// LS Electric XG5000 project: plc-assemble
// PLC LSPLC

PROGRAM NewProgram (task: 스캔 프로그램)

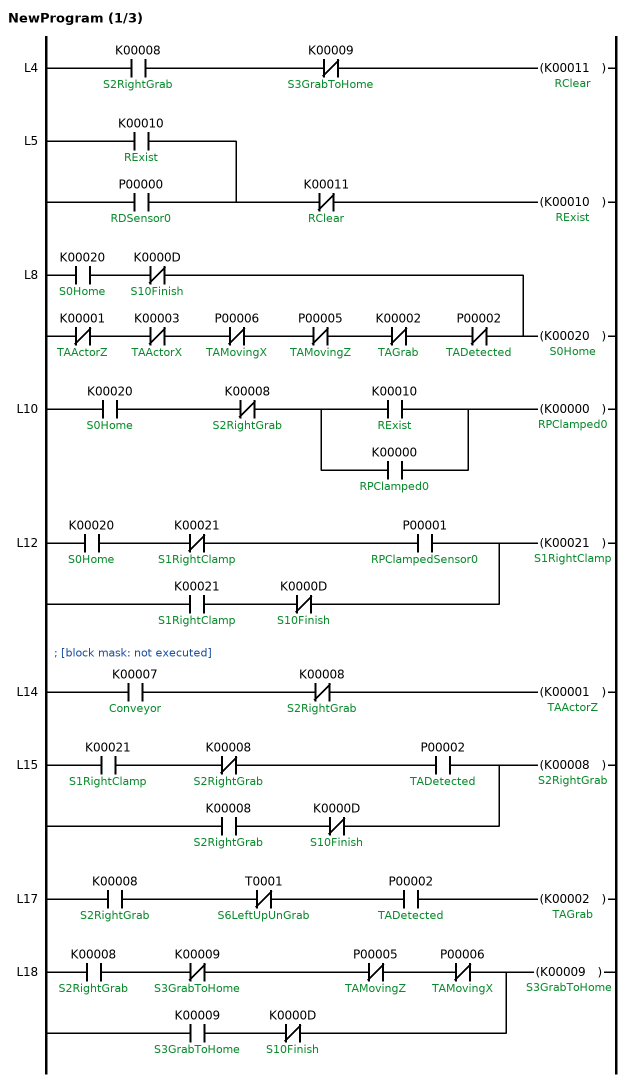
; L4
LOAD      K00008	// S2RightGrab
AND NOT   K00009	// S3GrabToHome
OUT       K00011	// RClear
; L5
LOAD      K00010	// RExist
OR        P00000	// RDSensor0
AND NOT   K00011	// RClear
OUT       K00010	// RExist
; L8
LOAD      K00020	// S0Home
AND NOT   K0000D	// S10Finish
LOAD NOT  K00001	// TAActorZ
AND NOT   K00003	// TAActorX
AND NOT   P00006	// TAMovingX
AND NOT   P00005	// TAMovingZ
AND NOT   K00002	// TAGrab
AND NOT   P00002	// TADetected
OR LOAD
OUT       K00020	// S0Home
; L10
LOAD      K00020	// S0Home
AND NOT   K00008	// S2RightGrab
LOAD      K00010	// RExist
OR        K00000	// RPClamped0
AND LOAD
OUT       K00000	// RPClamped0
; L12
LOAD      K00020	// S0Home
AND NOT   K00021	// S1RightClamp
AND       P00001	// RPClampedSensor0
LOAD      K00021	// S1RightClamp
AND NOT   K0000D	// S10Finish
OR LOAD
OUT       K00021	// S1RightClamp
; L14 (block mask: not executed)
LOAD      K00007	// Conveyor
AND NOT   K00008	// S2RightGrab
OUT       K00001	// TAActorZ
; L15
LOAD      K00021	// S1RightClamp
AND NOT   K00008	// S2RightGrab
AND       P00002	// TADetected
LOAD      K00008	// S2RightGrab
AND NOT   K0000D	// S10Finish
OR LOAD
OUT       K00008	// S2RightGrab
; L17
LOAD      K00008	// S2RightGrab
AND NOT   T0001	// S6LeftUpUnGrab
AND       P00002	// TADetected
OUT       K00002	// TAGrab
; L18
LOAD      K00008	// S2RightGrab
AND NOT   K00009	// S3GrabToHome
AND NOT   P00005	// TAMovingZ
AND NOT   P00006	// TAMovingX
LOAD      K00009	// S3GrabToHome
AND NOT   K0000D	// S10Finish
OR LOAD
OUT       K00009	// S3GrabToHome

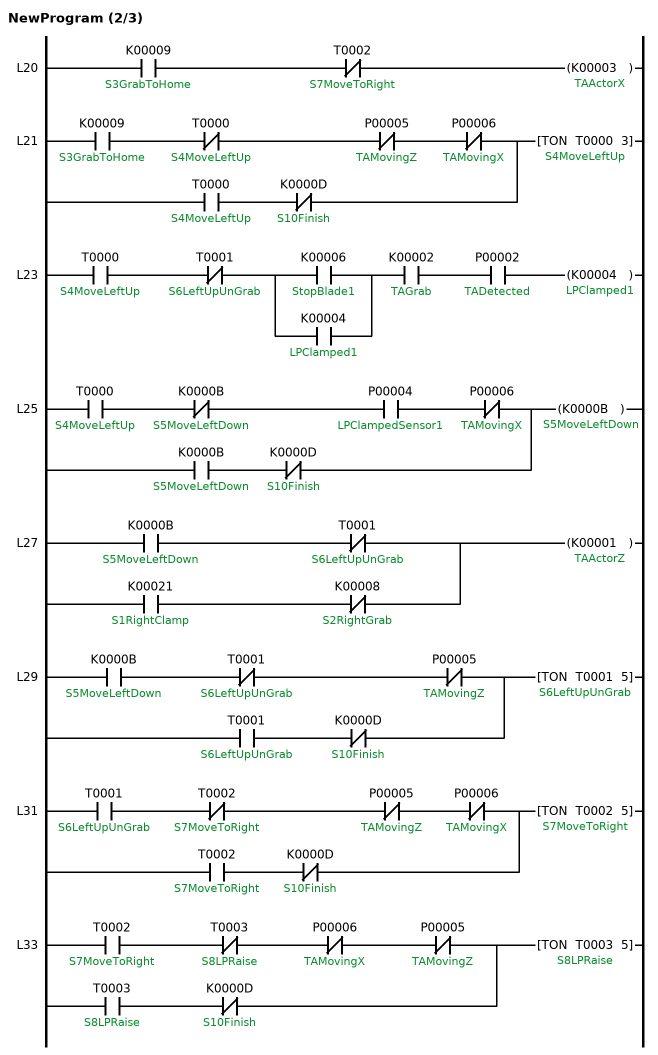
; L20
LOAD      K00009	// S3GrabToHome
AND NOT   T0002	// S7MoveToRight
OUT       K00003	// TAActorX
; L21
LOAD      K00009	// S3GrabToHome
AND NOT   T0000	// S4MoveLeftUp
AND NOT   P00005	// TAMovingZ
AND NOT   P00006	// TAMovingX
LOAD      T0000	// S4MoveLeftUp
AND NOT   K0000D	// S10Finish
OR LOAD
TON       T0000 3	// S4MoveLeftUp
; L23
LOAD      T0000	// S4MoveLeftUp
AND NOT   T0001	// S6LeftUpUnGrab
LOAD      K00006	// StopBlade1
OR        K00004	// LPClamped1
AND LOAD
AND       K00002	// TAGrab
AND       P00002	// TADetected
OUT       K00004	// LPClamped1
; L25
LOAD      T0000	// S4MoveLeftUp
AND NOT   K0000B	// S5MoveLeftDown
AND       P00004	// LPClampedSensor1
AND NOT   P00006	// TAMovingX
LOAD      K0000B	// S5MoveLeftDown
AND NOT   K0000D	// S10Finish
OR LOAD
OUT       K0000B	// S5MoveLeftDown
; L27
LOAD      K0000B	// S5MoveLeftDown
AND NOT   T0001	// S6LeftUpUnGrab
LOAD      K00021	// S1RightClamp
AND NOT   K00008	// S2RightGrab
OR LOAD
OUT       K00001	// TAActorZ
; L29
LOAD      K0000B	// S5MoveLeftDown
AND NOT   T0001	// S6LeftUpUnGrab
AND NOT   P00005	// TAMovingZ
LOAD      T0001	// S6LeftUpUnGrab
AND NOT   K0000D	// S10Finish
OR LOAD
TON       T0001 5	// S6LeftUpUnGrab
; L31
LOAD      T0001	// S6LeftUpUnGrab
AND NOT   T0002	// S7MoveToRight
AND NOT   P00005	// TAMovingZ
AND NOT   P00006	// TAMovingX
LOAD      T0002	// S7MoveToRight
AND NOT   K0000D	// S10Finish
OR LOAD
TON       T0002 5	// S7MoveToRight
; L33
LOAD      T0002	// S7MoveToRight
AND NOT   T0003	// S8LPRaise
AND NOT   P00006	// TAMovingX
AND NOT   P00005	// TAMovingZ
LOAD      T0003	// S8LPRaise
AND NOT   K0000D	// S10Finish
OR LOAD
TON       T0003 5	// S8LPRaise

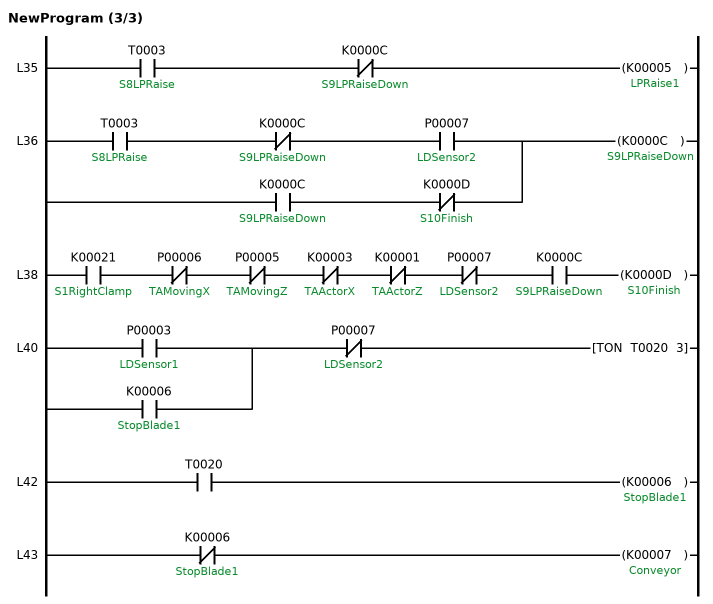
; L35
LOAD      T0003	// S8LPRaise
AND NOT   K0000C	// S9LPRaiseDown
OUT       K00005	// LPRaise1
; L36
LOAD      T0003	// S8LPRaise
AND NOT   K0000C	// S9LPRaiseDown
AND       P00007	// LDSensor2
LOAD      K0000C	// S9LPRaiseDown
AND NOT   K0000D	// S10Finish
OR LOAD
OUT       K0000C	// S9LPRaiseDown
; L38
LOAD      K00021	// S1RightClamp
AND NOT   P00006	// TAMovingX
AND NOT   P00005	// TAMovingZ
AND NOT   K00003	// TAActorX
AND NOT   K00001	// TAActorZ
AND NOT   P00007	// LDSensor2
AND       K0000C	// S9LPRaiseDown
OUT       K0000D	// S10Finish
; L40
LOAD      P00003	// LDSensor1
OR        K00006	// StopBlade1
AND NOT   P00007	// LDSensor2
TON       T0020 3
; L42
LOAD      T0020
OUT       K00006	// StopBlade1
; L43
LOAD NOT  K00006	// StopBlade1
OUT       K00007	// Conveyor